DATA_BLOCK "DB_DIH2_EX"
{ S7_Optimized_Access := 'FALSE' }
VERSION : 0.1
NON_RETAIN
   STRUCT
      TRIG : Int;   // Trigger signal 0-Waiting Trigger; 1-Trigger WProd 2-Trigger WPart; 3-Trigger Upt WS Status; 100-Err Write Ws; 101-Err Write Unit; Bussy-255
      Area : Struct
         Workstation : Struct
            "Name" : String[20];   // Workstation name
            State : String[20];   // Workstation state
            Attr_no_name : Array[1..10] of String[20];   // Attribute name to send for number format
            Attr_no_value : Array[1..10] of Int;   // Attribute numbers format
            Attr_txt_name : Array[1..5] of String[20];   // Attribute name to send for text format
            Attr_txt_value : Array[1..5] of String[20];   // Attribute text format
            Unit : Struct
               "Name" : String[20];   // Unit Name
               Attr_no_name : Array[1..10] of String[20];   // Attribute name to send for number format
               Attr_no_value : Array[1..10] of Int;   // Attribute numbers format
               Attr_txt_name : Array[1..5] of String[20];   // Attribute name to send for text format
               Attr_txt_value : Array[1..5] of String[20];   // Attribute text format
            END_STRUCT;
         END_STRUCT;
      END_STRUCT;
   END_STRUCT;


BEGIN

END_DATA_BLOCK

